// TIA Portal project "Farol_Estufagem" (V15)
// ..

(* hardware
DEVICE "S7-1200 station_1"  S7-1200 Station
   slot 0: "Rack_0"  S7-1200 Rack  Rack  V1.0
   slot 1: "PLC_1"  CPU 1212C DC/DC/DC  6ES7 212-1AE40-0XB0  V4.2
*)

// ===== PLC "PLC_1"  CPU 1212C DC/DC/DC =====
// protected blocks, not shown: "FB_Pisca_Pisca"

VAR_GLOBAL   // PLC tag table "Default tag table"
   "LAÇO 1" AT %I0.0 : Bool;
   "LAÇO 2" AT %I0.1 : Bool;
   "LAÇO 3" AT %I0.2 : Bool;
   "LACO_4" AT %I0.4 : Bool;
   "Botao_Sobe" AT %I0.7 : Bool;
   "VERDE PEDESTRE" AT %Q0.0 : Bool;
   "VERMELHO PEDESTRE" AT %Q0.1 : Bool;
   "VERDE CAMINHAO" AT %Q0.2 : Bool;
   "VERMELHO CAMINHAO" AT %Q0.3 : Bool;
   "Cancela" AT %Q0.5 : Bool;
   "System_Byte" AT %MB2 : Byte;
   "FirstScan" AT %M1.0 : Bool;
   "DiagStatusUpdate" AT %M1.1 : Bool;
   "AlwaysTRUE" AT %M1.2 : Bool;
   "AlwaysFALSE" AT %M1.3 : Bool;
   "Clock_Byte" AT %MB0 : Byte;
   "Clock_10Hz" AT %M0.0 : Bool;
   "Clock_5Hz" AT %M0.1 : Bool;
   "Clock_2.5Hz" AT %M0.2 : Bool;
   "Clock_2Hz" AT %M0.3 : Bool;
   "Clock_1.25Hz" AT %M0.4 : Bool;
   "Clock_1Hz" AT %M0.5 : Bool;
   "Clock_0.625Hz" AT %M0.6 : Bool;
   "Clock_0.5Hz" AT %M0.7 : Bool;
   "M0" AT %M10.0 : Bool;
   "M1" AT %M10.1 : Bool;
   "M2" AT %M10.2 : Bool;
   "M3" AT %M10.3 : Bool;
   "M4" AT %M10.4 : Bool;
   "M5" AT %M10.5 : Bool;
   "M6" AT %M10.6 : Bool;
   "M7" AT %M10.7 : Bool;
   "M8" AT %M11.0 : Bool;
   "M9" AT %M11.1 : Bool;
   "M10" AT %M11.2 : Bool;
   "M11" AT %M11.3 : Bool;
   "System_Byte(1)" AT %MB1 : Byte;
   "et" AT %MD4 : Time;
   "Pulso_1" AT %M3.0 : Bool;
   "Pulso_2" AT %M3.1 : Bool;
   "Pulso_3" AT %M3.2 : Bool;
   "Pulso_4" AT %M3.3 : Bool;
   "Pulso_5" AT %M3.4 : Bool;
   "M_Pulso" AT %M3.5 : Bool;
END_VAR

VAR_GLOBAL CONSTANT   // PLC tag table "Default tag table"
   "None(1)" : Pip := 65535;
   "Automatic update(1)" : Pip := 0;
   "PIP 1(1)" : Pip := 1;
   "PIP 2(1)" : Pip := 2;
   "PIP 3(1)" : Pip := 3;
   "PIP 4(1)" : Pip := 4;
   "PIP OB Servo(1)" : Pip := 32768;
   "Local~MC(1)" : Hw_SubModule := 51;
   "Local~Common(1)" : Hw_SubModule := 50;
   "Local~Device(1)" : Hw_Device := 32;
   "Local~Configuration(1)" : Hw_SubModule := 33;
   "Local~Exec(1)" : Hw_SubModule := 52;
   "Local(1)" : Hw_SubModule := 49;
   "Local~PROFINET_interface_1(1)" : Hw_Interface := 64;
   "Local~PROFINET_interface_1~Port_1(1)" : Hw_Interface := 65;
   "Local~HSC_1(1)" : Hw_Hsc := 257;
   "Local~HSC_2(1)" : Hw_Hsc := 258;
   "Local~HSC_3(1)" : Hw_Hsc := 259;
   "Local~HSC_4(1)" : Hw_Hsc := 260;
   "Local~HSC_5(1)" : Hw_Hsc := 261;
   "Local~HSC_6(1)" : Hw_Hsc := 262;
   "Local~AI_2_1(1)" : Hw_SubModule := 263;
   "Local~DI_14_DQ_10_1" : Hw_SubModule := 264;
   "Local~Pulse_1(1)" : Hw_Pwm := 265;
   "Local~Pulse_2(1)" : Hw_Pwm := 266;
   "Local~Pulse_3(1)" : Hw_Pwm := 267;
   "Local~Pulse_4(1)" : Hw_Pwm := 268;
   "OB_Main(1)" : OB_PCYCLE := 1;
END_VAR

DATA_BLOCK "Humble"   // DB1
{ S7_Optimized_Access := 'FALSE' }
VERSION : 0.1
   VAR
      Aciona_Farol : Bool;
   END_VAR
BEGIN
END_DATA_BLOCK

DATA_BLOCK "LogicaFarol_DB"   // DB3
{ S7_Optimized_Access := 'TRUE' }
VERSION : 0.1
// stored: InstanceOfName LogicaFarol
"LogicaFarol"
BEGIN
END_DATA_BLOCK

DATA_BLOCK "DB5_Pisca_Farol"   // DB5
{ S7_Optimized_Access := 'TRUE' }
VERSION : 0.1
// stored: InstanceOfName FB_Pisca_Farol
"FB_Pisca_Farol"
BEGIN
END_DATA_BLOCK

// folder: System blocks/Program resources

DATA_BLOCK "TP_Cancela"   // DB2
{ S7_Optimized_Access := 'TRUE' }
AUTHOR : Simatic
FAMILY : IEC
NAME : IEC_TMR
VERSION : 1.0
// stored: InstanceOfName IEC_TIMER
"IEC_TIMER"
BEGIN
END_DATA_BLOCK

DATA_BLOCK "IEC_Timer_0_DB_3"   // DB4
{ S7_Optimized_Access := 'TRUE' }
AUTHOR : Simatic
FAMILY : IEC
NAME : IEC_TMR
VERSION : 1.0
// stored: InstanceOfName IEC_TIMER
"IEC_TIMER"
BEGIN
END_DATA_BLOCK

// folder: (top level)

FUNCTION_BLOCK "LogicaFarol"   // FB1, LAD
{ S7_Optimized_Access := 'TRUE' }
VERSION : 0.1
   VAR_INPUT
      INLaco1 : Bool;   // Sinal do Laço 1.
      INLaco2 : Bool;   // Sinal do Laço 2.
      INLaco3 : Bool;   // Sinal do Laço 3.
   END_VAR
   VAR_OUTPUT
      OUTVerdePedestre : Bool;   // Sinal para o semaforo ligar verde para o pedestre.
      OUTVermelhoPedestre : Bool;   // Sinal para o semaforo ligar vermelho para o pedestre.
      OUTVerdeveiculo : Bool;   // Sinal para o semaforo ligar verde para o veiculo.
      OUTVermelhoveiculo : Bool;   // Sinal para o semaforo ligar vermelho para o veiculo.
   END_VAR
   VAR
      FiltroSinalLaco1 : TON_TIME;   // Temporizador para filtro do sinal do laço 1.
      FiltroSinalLaco2 : TON_TIME;   // Temporizador para filtro do sinal do laço 2.
      FiltroSinalLaco3 : TON_TIME;   // Temporizador para filtro do sinal do laço 3.
      ContagemCicloFarol : TP_TIME;   // Temporizador principal para contagem do ciclo do semaforo
      PulsoFiltroLaco1 : Bool;
      PulsoFiltroLaco2 : Bool;
      PulsoFiltroLaco3 : Bool;
   END_VAR
   VAR_TEMP   // added for the SCL form of the ladder/FBD networks
      _w1 : Bool;
      _w2 : Bool;
      _w3 : Bool;
   END_VAR
BEGIN

REGION Network 1: Filtro dos sinais dos laços de monitoramento do semaforo das docas.
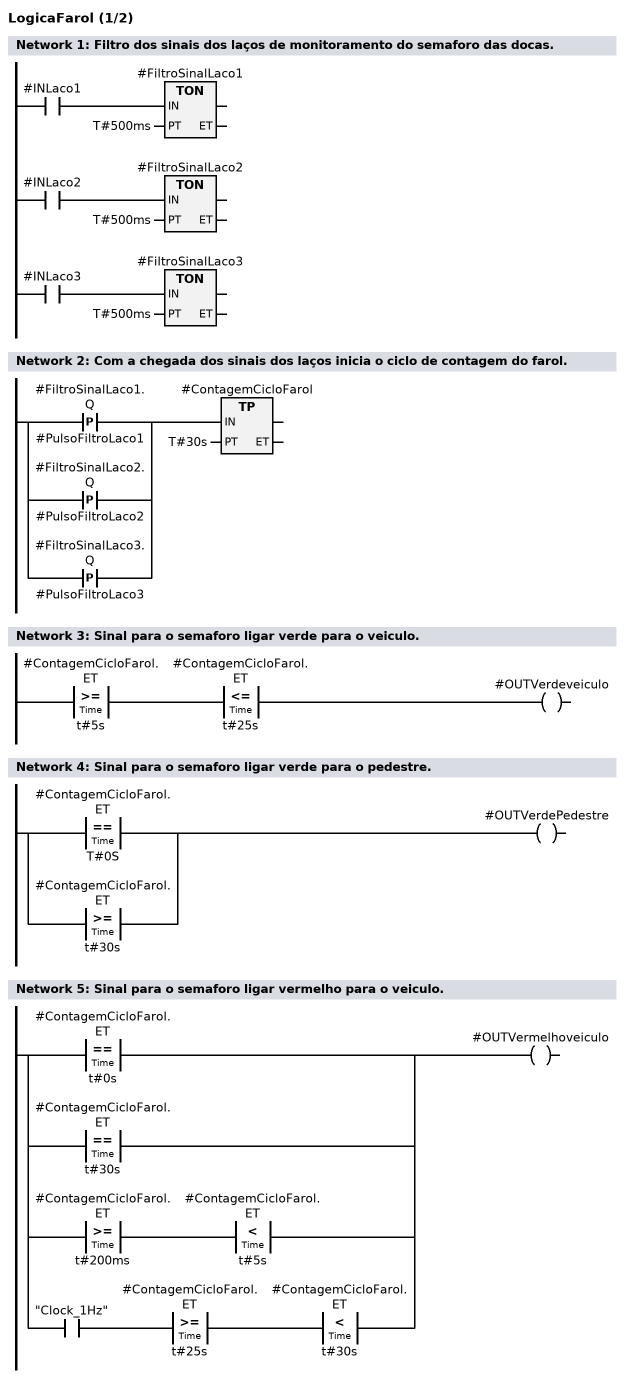
   #FiltroSinalLaco1(IN := #INLaco1, PT := T#500ms);   // TON
   #FiltroSinalLaco2(IN := #INLaco2, PT := T#500ms);   // TON
   #FiltroSinalLaco3(IN := #INLaco3, PT := T#500ms);   // TON
END_REGION

REGION Network 2: Com a chegada dos sinais dos laços inicia o ciclo de contagem do farol.
   #_w1 := #FiltroSinalLaco1.Q AND NOT #PulsoFiltroLaco1;   // rising edge of #FiltroSinalLaco1.Q
   #PulsoFiltroLaco1 := #FiltroSinalLaco1.Q;
   #_w2 := #FiltroSinalLaco2.Q AND NOT #PulsoFiltroLaco2;   // rising edge of #FiltroSinalLaco2.Q
   #PulsoFiltroLaco2 := #FiltroSinalLaco2.Q;
   #_w3 := #FiltroSinalLaco3.Q AND NOT #PulsoFiltroLaco3;   // rising edge of #FiltroSinalLaco3.Q
   #PulsoFiltroLaco3 := #FiltroSinalLaco3.Q;
   #ContagemCicloFarol(IN := #_w1 OR #_w2 OR #_w3, PT := T#30s);   // TP
END_REGION

REGION Network 3: Sinal para o semaforo ligar verde para o veiculo.
   RUNG wire#powerrail
      { S7_Templates := "SrcType := Time" } GE_Contact(in1 := #ContagemCicloFarol.ET, in2 := t#5s)
      { S7_Templates := "SrcType := Time" } LE_Contact(in1 := #ContagemCicloFarol.ET, in2 := t#25s)
      Coil( #OUTVerdeveiculo )
   END_RUNG
   // the same network as SCL:
   #OUTVerdeveiculo := (#ContagemCicloFarol.ET >= t#5s) AND (#ContagemCicloFarol.ET <= t#25s);
END_REGION

REGION Network 4: Sinal para o semaforo ligar verde para o pedestre.
   RUNG wire#powerrail
      { S7_Templates := "SrcType := Time" } EQ_Contact(in1 := #ContagemCicloFarol.ET, in2 := T#0S)
      wire#w1
      Coil( #OUTVerdePedestre )
   END_RUNG
   RUNG wire#powerrail
      { S7_Templates := "SrcType := Time" } GE_Contact(in1 := #ContagemCicloFarol.ET, in2 := t#30s)
   END_RUNG wire#w1
   // the same network as SCL:
   #OUTVerdePedestre := (#ContagemCicloFarol.ET = T#0S) OR (#ContagemCicloFarol.ET >= t#30s);
END_REGION

REGION Network 5: Sinal para o semaforo ligar vermelho para o veiculo.
   RUNG wire#powerrail
      { S7_Templates := "SrcType := Time" } EQ_Contact(in1 := #ContagemCicloFarol.ET, in2 := t#0s)
      wire#w1
      Coil( #OUTVermelhoveiculo )
   END_RUNG
   RUNG wire#powerrail
      { S7_Templates := "SrcType := Time" } EQ_Contact(in1 := #ContagemCicloFarol.ET, in2 := t#30s)
   END_RUNG wire#w1
   RUNG wire#powerrail
      { S7_Templates := "SrcType := Time" } GE_Contact(in1 := #ContagemCicloFarol.ET, in2 := t#200ms)
      { S7_Templates := "SrcType := Time" } LT_Contact(in1 := #ContagemCicloFarol.ET, in2 := t#5s)
   END_RUNG wire#w1
   RUNG wire#powerrail
      Contact( "Clock_1Hz" )
      { S7_Templates := "SrcType := Time" } GE_Contact(in1 := #ContagemCicloFarol.ET, in2 := t#25s)
      { S7_Templates := "SrcType := Time" } LT_Contact(in1 := #ContagemCicloFarol.ET, in2 := t#30s)
   END_RUNG wire#w1
   // the same network as SCL:
   #OUTVermelhoveiculo := (#ContagemCicloFarol.ET = t#0s) OR (#ContagemCicloFarol.ET = t#30s) OR ((#ContagemCicloFarol.ET >= t#200ms) AND (#ContagemCicloFarol.ET < t#5s)) OR ("Clock_1Hz" AND (#ContagemCicloFarol.ET >= t#25s) AND (#ContagemCicloFarol.ET < t#30s));
END_REGION

REGION Network 6: Sinal para o semaforo ligar vermelho para o pedestre.
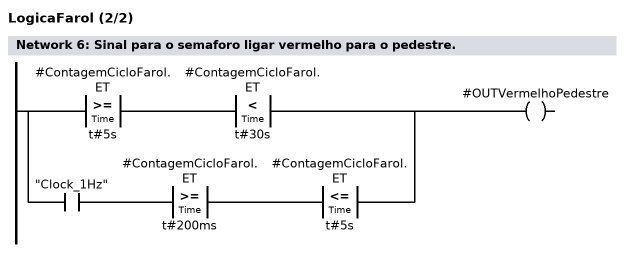
   RUNG wire#powerrail
      { S7_Templates := "SrcType := Time" } GE_Contact(in1 := #ContagemCicloFarol.ET, in2 := t#5s)
      { S7_Templates := "SrcType := Time" } LT_Contact(in1 := #ContagemCicloFarol.ET, in2 := t#30s)
      wire#w1
      Coil( #OUTVermelhoPedestre )
   END_RUNG
   RUNG wire#powerrail
      Contact( "Clock_1Hz" )
      { S7_Templates := "SrcType := Time" } GE_Contact(in1 := #ContagemCicloFarol.ET, in2 := t#200ms)
      { S7_Templates := "SrcType := Time" } LE_Contact(in1 := #ContagemCicloFarol.ET, in2 := t#5s)
   END_RUNG wire#w1
   // the same network as SCL:
   #OUTVermelhoPedestre := ((#ContagemCicloFarol.ET >= t#5s) AND (#ContagemCicloFarol.ET < t#30s)) OR ("Clock_1Hz" AND (#ContagemCicloFarol.ET >= t#200ms) AND (#ContagemCicloFarol.ET <= t#5s));
END_REGION
END_FUNCTION_BLOCK

FUNCTION_BLOCK "FB_Pisca_Farol"   // FB2, SCL
TITLE = Pisca_Farol
{ S7_Optimized_Access := 'TRUE' }
VERSION : 0.1
// Bloco responsavel por fazer o farol ficar piscante
   VAR_INPUT
      IN_Clock_1s : Bool;
   END_VAR
   VAR_OUTPUT
      OUT_Verde_Pedestre : Bool;   // Sinal para o semaforo ligar verde para o pedestre.
      OUT_Vermelho_Pedestre : Bool;   // Sinal para o semaforo ligar vermelho para o pedestre.
      OUT_Verde_Veiculo : Bool;   // Sinal para o semaforo ligar verde para o veiculo.
      OUT_Vermelho_Veiculo : Bool;   // Sinal para o semaforo ligar vermelho para o veiculo.
   END_VAR
   VAR
      M_Aux_Psica : Bool;
   END_VAR
BEGIN
   IF #IN_Clock_1s THEN
       #M_Aux_Psica := 1;
   ELSE
       #M_Aux_Psica := 0;
       ;
   END_IF;


    #OUT_Verde_Pedestre := NOT #M_Aux_Psica;
   #OUT_Verde_Veiculo := NOT #M_Aux_Psica;
   #OUT_Vermelho_Pedestre := #M_Aux_Psica;
   #OUT_Vermelho_Veiculo := #M_Aux_Psica;
END_FUNCTION_BLOCK

FUNCTION "FAROL" : Void   // FC1, LAD
{ S7_Optimized_Access := 'TRUE' }
VERSION : 0.1
   VAR_INPUT
      "LAÇO 1" : Bool;
      "LAÇO 2" : Bool;
      "LAÇO 3" : Bool;
   END_VAR
   VAR_OUTPUT
      "VERDE PEDESTRE" : Bool;
      "VERMELHO PEDESTRE" : Bool;
      "VERDE CAMINHAO" : Bool;
      "VERMELHO CAMINHAO" : Bool;
   END_VAR
   VAR_TEMP   // added for the SCL form of the ladder/FBD networks
      _w1 : Bool;
      _w2 : Bool;
      _w3 : Bool;
   END_VAR
BEGIN

REGION Network 1
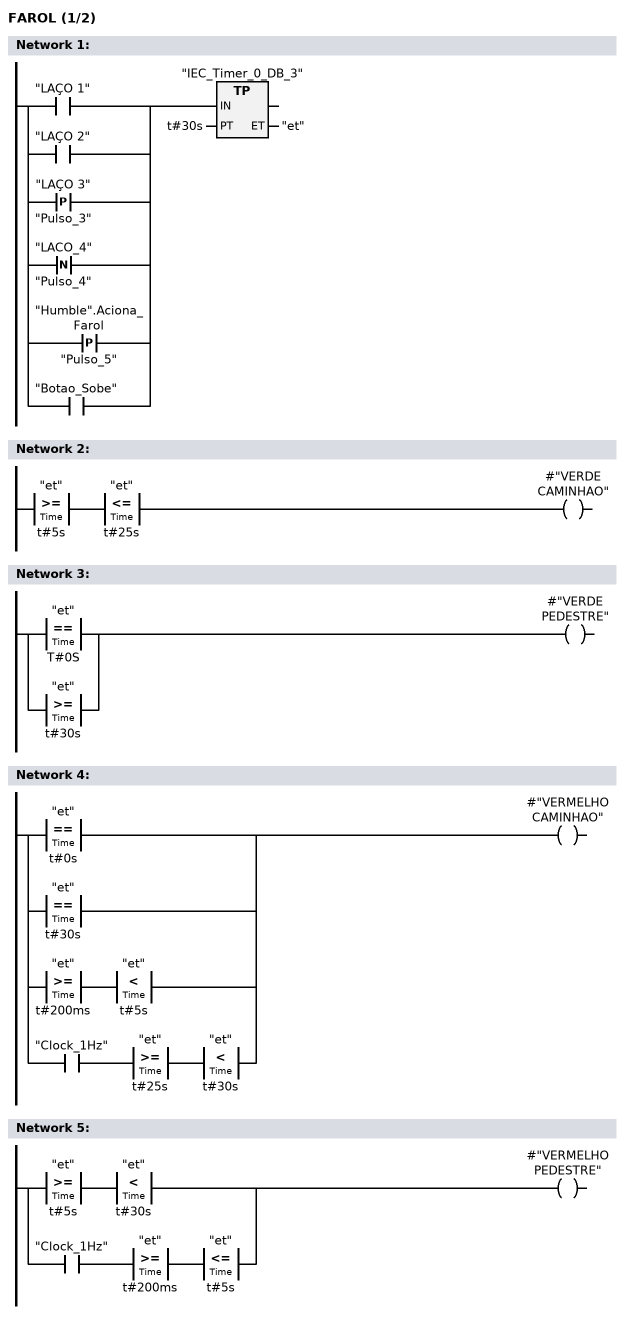
   #_w1 := "LAÇO 3" AND NOT "Pulso_3";   // rising edge of "LAÇO 3"
   "Pulso_3" := "LAÇO 3";
   #_w2 := NOT "LACO_4" AND "Pulso_4";   // falling edge of "LACO_4"
   "Pulso_4" := "LACO_4";
   #_w3 := "Humble".Aciona_Farol AND NOT "Pulso_5";   // rising edge of "Humble".Aciona_Farol
   "Pulso_5" := "Humble".Aciona_Farol;
   "IEC_Timer_0_DB_3".TP(IN := "LAÇO 1" OR "LAÇO 2" OR #_w1 OR #_w2 OR #_w3 OR "Botao_Sobe",
                         PT := t#30s,
                         ET => "et");
END_REGION

REGION Network 2
   RUNG wire#powerrail
      { S7_Templates := "SrcType := Time" } GE_Contact(in1 := "et", in2 := t#5s)
      { S7_Templates := "SrcType := Time" } LE_Contact(in1 := "et", in2 := t#25s)
      Coil( #"VERDE CAMINHAO" )
   END_RUNG
   // the same network as SCL:
   #"VERDE CAMINHAO" := ("et" >= t#5s) AND ("et" <= t#25s);
END_REGION

REGION Network 3
   RUNG wire#powerrail
      { S7_Templates := "SrcType := Time" } EQ_Contact(in1 := "et", in2 := T#0S)
      wire#w1
      Coil( #"VERDE PEDESTRE" )
   END_RUNG
   RUNG wire#powerrail
      { S7_Templates := "SrcType := Time" } GE_Contact(in1 := "et", in2 := t#30s)
   END_RUNG wire#w1
   // the same network as SCL:
   #"VERDE PEDESTRE" := ("et" = T#0S) OR ("et" >= t#30s);
END_REGION

REGION Network 4
   RUNG wire#powerrail
      { S7_Templates := "SrcType := Time" } EQ_Contact(in1 := "et", in2 := t#0s)
      wire#w1
      Coil( #"VERMELHO CAMINHAO" )
   END_RUNG
   RUNG wire#powerrail
      { S7_Templates := "SrcType := Time" } EQ_Contact(in1 := "et", in2 := t#30s)
   END_RUNG wire#w1
   RUNG wire#powerrail
      { S7_Templates := "SrcType := Time" } GE_Contact(in1 := "et", in2 := t#200ms)
      { S7_Templates := "SrcType := Time" } LT_Contact(in1 := "et", in2 := t#5s)
   END_RUNG wire#w1
   RUNG wire#powerrail
      Contact( "Clock_1Hz" )
      { S7_Templates := "SrcType := Time" } GE_Contact(in1 := "et", in2 := t#25s)
      { S7_Templates := "SrcType := Time" } LT_Contact(in1 := "et", in2 := t#30s)
   END_RUNG wire#w1
   // the same network as SCL:
   #"VERMELHO CAMINHAO" := ("et" = t#0s) OR ("et" = t#30s) OR (("et" >= t#200ms) AND ("et" < t#5s)) OR ("Clock_1Hz" AND ("et" >= t#25s) AND ("et" < t#30s));
END_REGION

REGION Network 5
   RUNG wire#powerrail
      { S7_Templates := "SrcType := Time" } GE_Contact(in1 := "et", in2 := t#5s)
      { S7_Templates := "SrcType := Time" } LT_Contact(in1 := "et", in2 := t#30s)
      wire#w1
      Coil( #"VERMELHO PEDESTRE" )
   END_RUNG
   RUNG wire#powerrail
      Contact( "Clock_1Hz" )
      { S7_Templates := "SrcType := Time" } GE_Contact(in1 := "et", in2 := t#200ms)
      { S7_Templates := "SrcType := Time" } LE_Contact(in1 := "et", in2 := t#5s)
   END_RUNG wire#w1
   // the same network as SCL:
   #"VERMELHO PEDESTRE" := (("et" >= t#5s) AND ("et" < t#30s)) OR ("Clock_1Hz" AND ("et" >= t#200ms) AND ("et" <= t#5s));
END_REGION

REGION Network 6
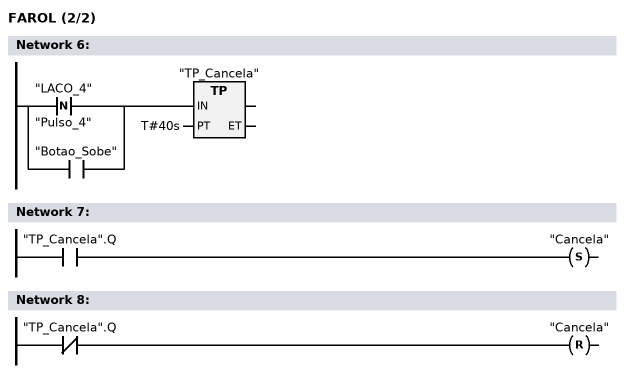
   #_w1 := NOT "LACO_4" AND "Pulso_4";   // falling edge of "LACO_4"
   "Pulso_4" := "LACO_4";
   "TP_Cancela".TP(IN := #_w1 OR "Botao_Sobe", PT := T#40s);
END_REGION

REGION Network 7
   RUNG wire#powerrail
      Contact( "TP_Cancela".Q )
      S_Coil( "Cancela" )
   END_RUNG
   // the same network as SCL:
   IF "TP_Cancela".Q THEN "Cancela" := TRUE; END_IF;
END_REGION

REGION Network 8
   RUNG wire#powerrail
      I_Contact( "TP_Cancela".Q )
      R_Coil( "Cancela" )
   END_RUNG
   // the same network as SCL:
   IF NOT "TP_Cancela".Q THEN "Cancela" := FALSE; END_IF;
END_REGION
END_FUNCTION

ORGANIZATION_BLOCK "Main"   // OB1, LAD, ProgramCycle
TITLE = "Main Program Sweep (Cycle)"
{ S7_Optimized_Access := 'TRUE' }
VERSION : 0.1
   VAR_INPUT
      Initial_Call : Bool;   // Initial call of this OB
      Remanence : Bool;   // =True, if remanent data are available
   END_VAR
BEGIN

REGION Network 1: LÓGICA PRINCIPAL PARA FINCIONAMENTO DO FAROL
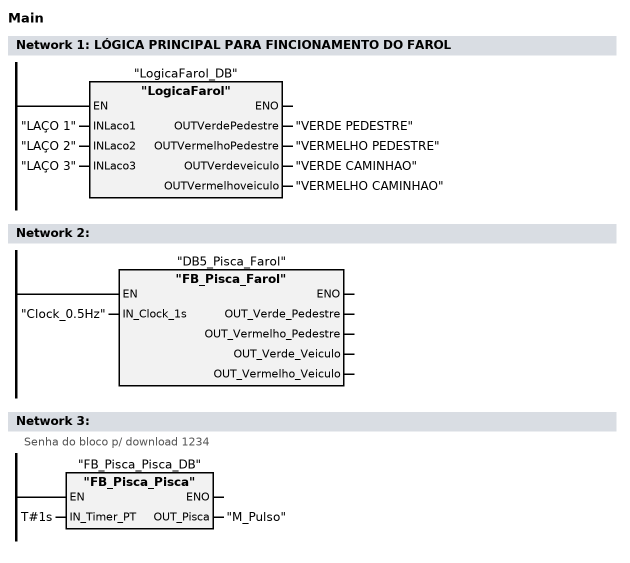
   RUNG wire#powerrail
      "LogicaFarol_DB"(INLaco1 := "LAÇO 1", INLaco2 := "LAÇO 2", INLaco3 := "LAÇO 3", OUTVerdePedestre => "VERDE PEDESTRE", OUTVermelhoPedestre => "VERMELHO PEDESTRE", OUTVerdeveiculo => "VERDE CAMINHAO", OUTVermelhoveiculo => "VERMELHO CAMINHAO")
   END_RUNG
   // the same network as SCL:
   "LogicaFarol_DB"(INLaco1 := "LAÇO 1",   // "LogicaFarol"
                    INLaco2 := "LAÇO 2",
                    INLaco3 := "LAÇO 3",
                    OUTVerdePedestre => "VERDE PEDESTRE",
                    OUTVermelhoPedestre => "VERMELHO PEDESTRE",
                    OUTVerdeveiculo => "VERDE CAMINHAO",
                    OUTVermelhoveiculo => "VERMELHO CAMINHAO");
END_REGION

REGION Network 2
   RUNG wire#powerrail
      "DB5_Pisca_Farol"(IN_Clock_1s := "Clock_0.5Hz", OUT_Verde_Pedestre =>, OUT_Vermelho_Pedestre =>, OUT_Verde_Veiculo =>, OUT_Vermelho_Veiculo =>)
   END_RUNG
   // the same network as SCL:
   "DB5_Pisca_Farol"(IN_Clock_1s := "Clock_0.5Hz");   // "FB_Pisca_Farol"
END_REGION

REGION Network 3
   // Senha do bloco p/ download 1234
   RUNG wire#powerrail
      "FB_Pisca_Pisca_DB"(IN_Timer_PT := T#1s, OUT_Pisca => "M_Pulso")
   END_RUNG
   // the same network as SCL:
   "FB_Pisca_Pisca_DB"(IN_Timer_PT := T#1s, OUT_Pisca => "M_Pulso");   // "FB_Pisca_Pisca"
END_REGION
END_ORGANIZATION_BLOCK